FUNCTION FC_7strConcatSeparator : T_DEFAULT_STR
VAR_INPUT
	iSeparator:		STRING := IING.STRING_UNDERSCORE;
	iStr1:			T_DEFAULT_STR;
	iStr2:			T_DEFAULT_STR;
	iStr3:			T_DEFAULT_STR;
	iStr4:			T_DEFAULT_STR;
	iStr5:			T_DEFAULT_STR;
	iStr6:			T_DEFAULT_STR;
	iStr7:			T_DEFAULT_STR;
END_VAR

FC_7strConcatSeparator := FC_2strConcatSeparator(iSeparator, FC_6strConcatSeparator(iSeparator, iStr1, iStr2, iStr3, iStr4, iStr5, iStr6), iStr7);

END_FUNCTION

(* stored: Version 1.1.0.1, ProductVersion 3.1.4026.18
   POU FC_7strConcatSeparator: Id {a9ec3cb1-8d11-4752-91d3-3edfa29c2943}, SpecialFunc None *)
